// TIA Portal V19 export
FUNCTION_BLOCK "An Scaling"   // FB5, LAD
{ S7_Optimized_Access := 'TRUE' }
// stored: MemoryReserve 100, SetENOAutomatically false
   VAR_INPUT
      "Sensor IN" : Int;
      "Analog Min" { ExternalAccessible := 'False'; ExternalVisible := 'False'; ExternalWritable := 'False'} : Int;
      "Analog Max" { ExternalAccessible := 'False'; ExternalVisible := 'False'; ExternalWritable := 'False'} : Int;
      "Scaled Min" { ExternalAccessible := 'False'; ExternalVisible := 'False'; ExternalWritable := 'False'} : Real;
      "Scaled Max" { ExternalAccessible := 'False'; ExternalVisible := 'False'; ExternalWritable := 'False'} : Real;
   END_VAR
   VAR_OUTPUT
      Scaled_Sensor : Real;
   END_VAR
   VAR
      Normalised_sensor { ExternalAccessible := 'False'; ExternalVisible := 'False'; ExternalWritable := 'False'} : Real;
      sensor_result { ExternalAccessible := 'False'; ExternalVisible := 'False'; ExternalWritable := 'False'} : Int;
   END_VAR
BEGIN

REGION Network 1: scale the sensor
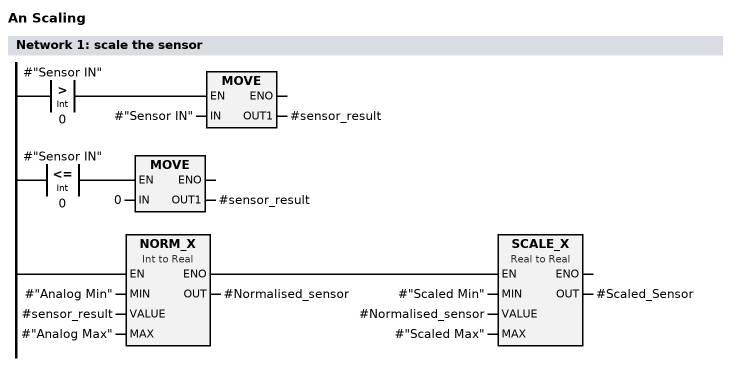
   RUNG wire#powerrail
      { S7_Templates := "SrcType := Int" } GT_Contact(in1 := #"Sensor IN", in2 := 0)
      { S7_GenerateENO := "TRUE" } Move(in := #"Sensor IN", out1 => #sensor_result)
   END_RUNG
   RUNG wire#powerrail
      { S7_Templates := "SrcType := Int" } LE_Contact(in1 := #"Sensor IN", in2 := 0)
      { S7_GenerateENO := "TRUE" } Move(in := 0, out1 => #sensor_result)
   END_RUNG
   RUNG wire#powerrail
      { S7_Templates := "[SrcType := Int, DestType := Real]"; S7_GenerateENO := "TRUE" } Normalize(min := #"Analog Min", value := #sensor_result, max := #"Analog Max", out => #Normalised_sensor)
      { S7_Templates := "[SrcType := Real, DestType := Real]"; S7_GenerateENO := "TRUE" } Scale(min := #"Scaled Min", value := #Normalised_sensor, max := #"Scaled Max", out => #Scaled_Sensor)
   END_RUNG
   // the same network as SCL:
   // ENO of a box is taken as its EN; it also drops when the box reports an error
   IF #"Sensor IN" > 0 THEN #sensor_result := #"Sensor IN"; END_IF;
   IF #"Sensor IN" <= 0 THEN #sensor_result := 0; END_IF;
   #Normalised_sensor := NORM_X(MIN := #"Analog Min", VALUE := #sensor_result, MAX := #"Analog Max");
   #Scaled_Sensor := SCALE_X(MIN := #"Scaled Min", VALUE := #Normalised_sensor, MAX := #"Scaled Max");
END_REGION
END_FUNCTION_BLOCK
